INTERFACE ICrud

METHOD Create : TcoCore.ITcoTaskStatus
VAR_INPUT
	Identifier : STRING(255);
END_VAR
END_METHOD

METHOD Delete : TcoCore.ITcoTaskStatus
VAR_INPUT
	Identifier : STRING(255);
END_VAR
END_METHOD

METHOD Read : TcoCore.ITcoTaskStatus
VAR_INPUT
	Identifier : STRING(255);
END_VAR
END_METHOD

METHOD Update : TcoCore.ITcoTaskStatus
VAR_INPUT
	Identifier : STRING(255);
END_VAR
END_METHOD

END_INTERFACE

(* stored: Version 1.1.0.1, ProductVersion 3.1.4024.6
   Itf ICrud: Id {5f3c65e2-780e-08d0-1226-02e7fb1c5c1d}
   Method Create: Id {0515119d-8a26-0ad7-1ffa-08bce7e22829}
   Method Delete: Id {21cbb8cb-d3c3-0ef6-0dbc-3fd4191b36ee}
   Method Read: Id {56192ca7-8514-0978-1e5e-6ff33827c9c4}
   Method Update: Id {62ce4dd0-f7ce-0347-3989-565f1358c0bb} *)
